{attribute 'qualified_only'}
{attribute 'strict'}
TYPE ControllerState :
(
	init 			:= 0,
	idle			:= 1,
	calcTrajectory 	:= 2,
	setTrajectory	:= 3,
	ready			:= 4,
	driving			:= 5

);
END_TYPE

(* stored: Version 1.1.0.1, ProductVersion 3.1.4024.11
   DUT ControllerState: Id {807775c5-1a7b-4f15-a7de-7f752c544cb4} *)
